KUKA KRL program: Sps2.sub

&ACCESS RV
&PARAM TPVW_VERSION=8.3.18
DEF  SPS2 ( )
; FOLD ;%{H} %MKUKATPVW
;Init part of vw_usr_s
VW_USR_S (#USR_INIT_SUB2)

LOOP
;Freilaufende SPS
MAKROSUBMIT2()

WAIT FOR NOT $POWER_FAIL
ENDLOOP
END
;ENDFOLD
